FUNCTION_BLOCK FB_CameraDummy EXTENDS FB_CameraBase
VAR_INPUT
END_VAR
VAR_OUTPUT
END_VAR
VAR
END_VAR

{attribute 'monitoring':='call'}
PROPERTY eCameraMode : E_CameraMode
GET
eCameraMode := _eCameraMode;
IF _eCameraMode = E_CameraMode.Auto THEN
  eCameraMode := E_CameraMode.NoCorrection;
END_IF
END_GET
END_PROPERTY

PROPERTY eDeviceType : E_CameraDevice
GET
eDeviceType := E_CameraDevice.SheetDetect;
END_GET
END_PROPERTY

METHOD GetCamStatus : BOOL
VAR_OUTPUT
  bConnectionOK  : BOOL;    // Camera connected
  bTeachOk       : BOOL;    // Teach successful
  nTeachedPoints : UDINT;   // Teached points for this job
  nScannedPoints : UDINT;   // Scanned points on current sheet
  bCamStarted    : BOOL;    // Camera trigger is active, cam started
  bCamDone       : BOOL;    // Camera finished on last CT
  bErrors        : ARRAY[1..GVL_Camera.nC_NbCamErrors] OF BOOL;  // generic error flag list
END_VAR
bConnectionOK  := TRUE;  //NO comm with a cam 
bTeachOk       := TRUE;  //NO teach availabe
nTeachedPoints := 0;
nScannedPoints := 0;
bCamStarted    := _bCamStarted;
bCamDone       := _bCamDone;

GetCamStatus := TRUE;
END_METHOD

(*
  Set mode to camera.
  :return: TRUE if success
*)
METHOD setCameraMode : BOOL
VAR_INPUT
  eCameraMode : E_CameraMode;
END_VAR
IF eCameraMode = E_CameraMode.NoCorrection THEN   // supported mode
  
  _eCameraMode := eCameraMode; 
  setCameraMode := TRUE;        // set desired mode
ELSE
  LogError(F_Concat3('Camera mode=', TO_STRING(eCameraMode), ' not supported by camera'));
  _eCameraMode := E_CameraMode.NoCorrection;
END_IF
END_METHOD

{attribute 'monitoring':='variable'}
PROPERTY sName : STRING
GET
sName := 'SheetDetect';
END_GET
END_PROPERTY

END_FUNCTION_BLOCK

(* stored: Version 1.1.0.1, ProductVersion 3.1.4024.3
   POU FB_CameraDummy: Id {fb042f63-d6eb-4556-94a2-674fae320829}, SpecialFunc None
   Property eCameraMode: Id {53cb1655-e0b5-4df5-82cf-8e993d9ee019}
   Get Get: Id {ccab4305-c3f0-406a-b402-36c608c04c35}
   Property eDeviceType: Id {23a50069-69d1-4e0c-baa6-252c56a81b22}
   Get Get: Id {5f28284e-32a0-4fdd-899e-8ce443075433}
   Method GetCamStatus: Id {2242ecf5-8c2b-4177-a249-a9c70a4011bb}
   Method setCameraMode: Id {faf52507-a55c-4852-a33b-a6a7ec32731d}
   Property sName: Id {47709119-4c99-45dd-8ef0-7c2b3c4235a6}
   Get Get: Id {a8946bb1-709d-4530-b955-95040efca2b0} *)
